PROGRAM MAIN
VAR
END_VAR

END_PROGRAM

(* stored: Version 1.1.0.1
   POU MAIN: Id {d51c8b77-0651-4e7e-9856-5a5d0fda5dc4} *)
